TYPE ProcessModulesConfig :
STRUCT
	PsdConfig : PsdConfig;
	LightspeedConfig : LightspeedConfig;	
	NstConfig : NstConfig;
	PhotoLumConfig : PhotoLumConfig;
END_STRUCT
END_TYPE

(* stored: Version 1.1.0.1, ProductVersion 3.1.4024.12
   DUT ProcessModulesConfig: Id {bc8a1c40-80c7-4cd2-a1ec-24c97966910f} *)
